// TIA Portal V16 export
// export: Created 2021-08-30T11:09:34.6105891Z, ExportSetting WithDefaults, DisplayName Totally Integrated Automation Portal, DisplayVersion V16 Update 3, DisplayName TIA Portal Version Control Interface, DisplayVersion V16 Update 2, DisplayName TIA Portal Openness, DisplayVersion V16 Update 3, DisplayName TIA Portal Teamcenter Gateway, DisplayVersion V16, DisplayName STEP 7 Professional, DisplayVersion V16 Update 3, DisplayName STEP 7 Safety, DisplayVersion V16, DisplayName WinCC Advanced, DisplayVersion V16 Update 3
DATA_BLOCK "dtPump"   // DB4
{ S7_Optimized_Access := 'FALSE' }
VERSION : 0.1
// stored: AutoNumber true, DBAccessibleFromOPCUA true, IsOnlyStoredInLoadMemory false, IsWriteProtectedInAS false
   VAR RETAIN
      P301 : "Pump";
      P302 { S7_SetPoint := 'True'} : "Pump";
      P1201 { S7_SetPoint := 'True'} : "Pump";
      P1202 { S7_SetPoint := 'True'} : "Pump";
   END_VAR
BEGIN
END_DATA_BLOCK
